FUNCTION_BLOCK IA_WBSD (* ISOBUS Adapter for Wheel Based Speed and Distance (WBSD) *)
  (* Standard: ISO 11783-7; Classification: PGN 65096; Description: Copyright (c) 2024 HR Agrartechnik GmbH This program and the accompanying materials are made available under the terms of the Eclipse Public License 2.0 which is available at https://www.eclipse.org/legal/epl-2.0/ SPDX-License-Identifier: EPL-2.0 *)
  (* Version 1.3, 2026-09-17, Franz Höpfinger, HR Agrartechnik GmbH, Bugfix (Franz: 'IA_VDS hat einen Bug, moeglicherweise alle anderen auch'): .IND->TIMEOUT.E1 ergaenzt (analog IA_VDS) - bisher wurde TIMEOUT.E1 NUR von .TIMEOUT gefeuert (Timeout-Beginn), nie beim Eintreffen einer normalen Botschaft (.IND) - TIMEOUT.D1 (Q_timeout=FALSE) wurde also gesetzt, aber nie an den TIMEOUT-Plug propagiert, sobald der Timeout wieder endete. *)
  (* Version 1.2, 2026-09-16, Franz Höpfinger, HR Agrartechnik GmbH, E_D_FF_ANY-Aenderungsfilter fuer SPEED/DISTANCE ergaenzt (analog IA_RPTO v1.1). *)
  (* Version 1.1, 2026-04-19, Franz Höpfinger, HR Agrartechnik GmbH, Fixed: Use conversion blocks to properly connect internal pins to adapter plugs *)
  (* Version 1.0, 2026-04-19, Franz Höpfinger, HR Agrartechnik GmbH, initial API and implementation (Adapter Wrapper for I_WBSD) *)
  PACKAGE isobus::tecu;
  (* Documentation:
  ISOBUS Adapter for Wheel Based Speed and Distance (WBSD)
   TIMEOUT.E1-Verdrahtung: I_WBSD.TIMEOUT (echter Timeout-Eintritt) UND I_WBSD.IND (Normalbetrieb) sind beide auf den Adapter-Plug TIMEOUT.E1 verdrahtet - bewusst so, damit TIMEOUT.D1 (Q_timeout) am Adapter-Plug auch beim Zuruecksetzen auf false aktualisiert wird, nicht nur beim Eintreten des Timeouts. Der zugrundeliegende TIMEOUT/IND-Vertrag von I_WBSD selbst ist in dessen eigener .fbt-Datei dokumentiert.
  *)
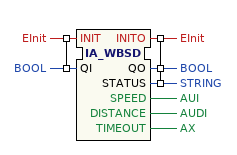
  EVENT_INPUT
    INIT : EInit WITH QI; (* Service Initialization *)
  END_EVENT
  EVENT_OUTPUT
    INITO : EInit WITH QO, STATUS; (* Initialization Confirm *)
  END_EVENT
  VAR_INPUT
    QI : BOOL; (* Event Input Qualifier *)
  END_VAR
  VAR_OUTPUT
    QO : BOOL; (* Event Output Qualifier *)
    STATUS : STRING;
  END_VAR
  PLUGS
    SPEED : adapter::types::unidirectional::AUI; (* Wheel-based machine speed *)
    DISTANCE : adapter::types::unidirectional::AUDI; (* Wheel-based machine distance *)
    TIMEOUT : adapter::types::unidirectional::AX; (* Timeout Status *)
  END_PLUGS
  FBS
    I_WBSD : isobus::tecu::I_WBSD;
    E_D_FF_Speed : iec61499::events::E_D_FF_ANY;
    E_D_FF_Distance : iec61499::events::E_D_FF_ANY;
  END_FBS
  EVENT_CONNECTIONS
    INIT TO I_WBSD.INIT;
    I_WBSD.INITO TO INITO;
    I_WBSD.TIMEOUT TO TIMEOUT.E1;
    I_WBSD.IND TO E_D_FF_Distance.CLK;
    E_D_FF_Distance.EO TO DISTANCE.E1;
    I_WBSD.IND TO E_D_FF_Speed.CLK;
    E_D_FF_Speed.EO TO SPEED.E1;
    I_WBSD.IND TO TIMEOUT.E1;
  END_CONNECTIONS
  DATA_CONNECTIONS
    QI TO I_WBSD.QI;
    I_WBSD.QO TO QO;
    I_WBSD.STATUS TO STATUS;
    I_WBSD.Q_timeout TO TIMEOUT.D1;
    I_WBSD.WHEELBASEDMACHINESPEED TO E_D_FF_Speed.D;
    E_D_FF_Speed.Q TO SPEED.D1;
    I_WBSD.WHEELBASEDMACHINEDISTANCE TO E_D_FF_Distance.D;
    E_D_FF_Distance.Q TO DISTANCE.D1;
  END_CONNECTIONS
END_FUNCTION_BLOCK
